// Enumerator contains packml state, unfortunatly named status
{attribute 'qualified_only'}
{attribute 'strict'}
TYPE E_Status :
(
	undefined:=0,
	clearing,
	stopped,
	starting,
	idle,
	suspended,
	execute,
	stopping,
	aborting,
	aborted,
	holding,
	held,
	unholding,
	suspending,
	unsuspending,
	resetting,
	completing,
	completed
);
END_TYPE

(* stored: Version 1.1.0.1, ProductVersion 3.1.4024.12
   DUT E_Status: Id {02e5105c-7e33-4838-8848-6543bca7cf3f} *)
